TYPE ST_ReceivedData :
STRUCT
	name :STRING;
	zipball_url :STRING;
	tarball_url :STRING;
END_STRUCT
END_TYPE

(* stored: Version 1.1.0.1, ProductVersion 3.1.4024.6
   DUT ST_ReceivedData: Id {4d061561-f78a-4b91-bcf9-7c79fb3a7d37} *)
